FUNCTION_BLOCK FB_Stewart
VAR_INPUT

END_VAR
VAR_OUTPUT

END_VAR
VAR
	txData				: TxStewart;
	rxData				: RxStewart;
	
	ipAddr 				: UDINT;
	remotePort 			: UINT;
	localPort 			: UINT;
	
	udpClient 			: FB_UdpClient(ipAddr, remotePort, localPort, SIZEOF(txData), ADR(txData), SIZEOF(rxData), ADR(rxData));
	
	pi					: REAL := 3.141592653589793;
	
END_VAR



// Update counter
txData.COUNT := txData.COUNT + 1;

// Exhange data using UDP connection
udpClient();

METHOD FB_init : BOOL
VAR_INPUT
	bInitRetains : BOOL; // if TRUE, the retain variables are initialized (warm start / cold start)
	bInCopyCode : BOOL;  // if TRUE, the instance afterwards gets moved into the copy code (online change)
	
	// Contructor arguments
	_ipAddr 			: UDINT;
	_remotePort 		: UINT;
	_localPort 		: UINT;
END_VAR
// Initilize parameters
ipAddr := _ipAddr;
remotePort := _remotePort;
localPort := _localPort;

// Construct FB_UdpClient
udpClient.FB_init(bInitRetains, bInCopyCode, ipAddr, remotePort, localPort, SIZEOF(txData), ADR(txData), SIZEOF(rxData), ADR(rxData));
END_METHOD

END_FUNCTION_BLOCK

(* stored: Version 1.1.0.1, ProductVersion 3.1.4020.12
   POU FB_Stewart: Id {c939fb9b-18fc-49a0-acdf-554ae7fa888b}, SpecialFunc None
   Method FB_init: Id {4975fdc8-91bb-4f8a-803d-234e9d5a5bf6} *)
